TEXTLIST languages
  0 = '英語'
  1 = '日本語'
   = ''
END_TEXTLIST

(* stored: Version 1.1.0.1
   TextList languages: Id {d7e57922-d902-472f-b5de-84089fe91c0a} *)
